(* CoDeSys 2.3 export: ST_TACK_VALVE_CFG.EXP *)

(* Data type *)
TYPE ST_TACK_VALVE_CFG :
STRUCT
	Cycle   : REAL; (*Seconds*)
	TimeMax : REAL; (*Seconds*)

	Hyst_HeelH : REAL;
	Hyst_HeelL : REAL;
	Hyst_Time  : REAL;	(*Seconds*)

END_STRUCT
END_TYPE
